// TwinCAT 3 PLC project green_crane
// ProgramVersion: 3.1.4026.19
// libraries:
//   Tc2_Standard, * (Beckhoff Automation GmbH)
//   Tc2_System, * (Beckhoff Automation GmbH)
// project tree:
//   Control/ AB_baseController.TcPOU, FB_AutoControl.TcPOU, FB_manualControl.TcPOU, I_craneControl.TcIO
//   DUTs/ E_CraneModes.TcDUT, E_CraneStatus.TcDUT
//   IOinterface/ FB_ioSim.TcPOU, I_ioInterface.TcIO
//   / PlcTask.TcTTO, simTask.TcTTO
//   POUs/ F_CalcAngle.TcPOU, F_stateMachine.TcPOU, MAIN.TcPOU, ST_inputs_analog.TcDUT, ST_in_digital.TcDUT, ST_ValvePos.TcDUT
//   Simulator/ FB_CylinderSimulator.TcPOU, P_Simulator.TcPOU
// real-time tasks:
//   TASK PlcTask: cycle T#10ms, priority 20, ADS port 350
//   TASK simTask: cycle T#100us, priority 1, ADS port 351

CONFIGURATION green_crane
    RESOURCE PLC ON TwinCAT3
        TASK PlcTask(INTERVAL := T#10ms, PRIORITY := 20);
        TASK simTask(INTERVAL := T#100us, PRIORITY := 1);
        PROGRAM MAIN WITH PlcTask : MAIN;
        PROGRAM P_Simulator WITH simTask : P_Simulator;
    END_RESOURCE
END_CONFIGURATION

// ---- DUTs/E_CraneModes.TcDUT
{attribute 'qualified_only'}
{attribute 'strict'}
{attribute 'to_string'}
TYPE E_CraneModes :
(
	Manual := 0,
	Auto := 1
);
END_TYPE

// ---- DUTs/E_CraneStatus.TcDUT
{attribute 'qualified_only'}
{attribute 'strict'}
{attribute 'to_string'}
TYPE E_CraneStatus :
(
	Off := 0,
	On := 1,
	Ready := 2,
	Running := 3
);
END_TYPE

// ---- POUs/ST_inputs_analog.TcDUT
TYPE ST_inputs_analog :
STRUCT	
	fJoystick : LREAL;
	fPistonPos : LREAL; // [mm] crane piston position
	fP_piston : LREAL; // [bar]
	fP_rod : LREAL; // [bar]
END_STRUCT
END_TYPE

// ---- POUs/ST_in_digital.TcDUT
TYPE ST_in_digital :
STRUCT
	bCranePower : BOOL := FALSE;
	bStartCrane : BOOL := FALSE;
	bEnableCraneMotion : BOOL := FALSE;
	eModeSwitch : E_CraneModes;
END_STRUCT
END_TYPE

// ---- POUs/ST_ValvePos.TcDUT
TYPE ST_ValvePos :
STRUCT
	rCylinderValve : REAL;
END_STRUCT
END_TYPE

// ---- Control/I_craneControl.TcIO
INTERFACE I_craneControl
VAR_INPUT
END_VAR
VAR_OUTPUT
END_VAR

METHOD control_crane
VAR_INPUT
	stInputs : ST_inputs_analog;
END_VAR
VAR_OUTPUT
	fCylValve : REAL;
END_VAR
END_METHOD

METHOD controller
VAR_INPUT
	stButtonInputs : ST_in_digital;
	stAnalogInputs : ST_inputs_analog;
END_VAR
VAR_OUTPUT
	stOutput : ST_ValvePos;
END_VAR
END_METHOD

END_INTERFACE

// ---- IOinterface/I_ioInterface.TcIO
INTERFACE I_ioInterface

METHOD getOutputs
VAR_IN_OUT
	stSimOut : ST_inputs_analog;
END_VAR
END_METHOD

METHOD setInputs
VAR_INPUT
	stValvePos	: ST_ValvePos;
	eCraneState : E_CraneStatus;
END_VAR
END_METHOD

END_INTERFACE

// ---- POUs/MAIN.TcPOU
PROGRAM MAIN
VAR
	stButtonInputs : ST_in_digital;
	stAnalogInputs : ST_inputs_analog;
	stOutputs : ST_ValvePos;
	eCraneMode : E_CraneStatus;
	ipControlMode : I_craneControl;
	fbManual : FB_manualControl;
	fbAuto : FB_AutoControl;
	stValveOut : ST_ValvePos;
	fbIOsim : FB_ioSim;
	fBoomAng : LREAL;
	fBoomAngRef : LREAL;
END_VAR

eCraneMode := F_stateMachine(stButtonInputs);
CASE stButtonInputs.eModeSwitch OF //polymorphism using interface pointer ipControlMode
		E_CraneModes.Manual:
			ipControlMode := fbManual;
		E_CraneModes.Auto:
			ipControlMode := fbAuto;
END_CASE

IF eCraneMode = E_CraneStatus.Running AND ipControlMode <> 0  THEN
	fbIOsim.getOutputs(stSimOut := stAnalogInputs);
	ipControlMode.controller(stButtonInputs := stButtonInputs,
		stAnalogInputs := stAnalogInputs,
		stOutput => stValveOut);
	fbIOsim.setInputs(stValvePos := stValveOut,
		eCraneState := eCraneMode);
END_IF

fBoomAng := F_CalcAngle(stAnalogInputs.fPistonPos);

END_PROGRAM

// ---- Control/FB_manualControl.TcPOU
FUNCTION_BLOCK FB_manualControl EXTENDS AB_baseController
VAR_INPUT
END_VAR
VAR_OUTPUT
END_VAR
VAR
END_VAR

METHOD control_winch
VAR_INPUT
	stInputs	: ST_inputs_analog;
END_VAR
VAR_OUTPUT
	fMotorValve	: REAL;
END_VAR
fMotorValve := -1.0;
END_METHOD

END_FUNCTION_BLOCK

// ---- Control/AB_baseController.TcPOU
FUNCTION_BLOCK ABSTRACT AB_baseController IMPLEMENTS I_craneControl
VAR_INPUT
END_VAR
VAR_OUTPUT
END_VAR
VAR
END_VAR

METHOD ABSTRACT control_crane 
VAR_INPUT
	stInputs	: ST_inputs_analog;
END_VAR
VAR_OUTPUT
	fCylValve	: REAL;
END_VAR
END_METHOD

METHOD controller
VAR_INPUT
	stButtonInputs	: ST_in_digital;
	stAnalogInputs	: ST_inputs_analog;
END_VAR
VAR_OUTPUT
	stOutput	: ST_ValvePos;
END_VAR
stOutput.rCylinderValve := control_crane(stInputs := stAnalogInputs);
END_METHOD

END_FUNCTION_BLOCK

// ---- Control/FB_AutoControl.TcPOU
FUNCTION_BLOCK FB_AutoControl EXTENDS AB_baseController
VAR_INPUT
END_VAR
VAR_OUTPUT
END_VAR
VAR
END_VAR

METHOD control_crane
VAR_INPUT
	stInputs	: ST_inputs_analog;
END_VAR
VAR_OUTPUT
	fCylValve	: REAL;
END_VAR
fCylValve := 0;
END_METHOD

END_FUNCTION_BLOCK

// ---- IOinterface/FB_ioSim.TcPOU
FUNCTION_BLOCK PUBLIC FB_ioSim IMPLEMENTS I_ioInterface
VAR_INPUT
END_VAR
VAR_OUTPUT
END_VAR
VAR
END_VAR

METHOD getOutputs
VAR_IN_OUT
	stSimOut : ST_inputs_analog;
END_VAR
stSimOut.fP_piston := P_Simulator.stSimSystemOutputs.fP_piston;
stSimOut.fP_rod := P_Simulator.stSimSystemOutputs.fP_rod;
stSimOut.fPistonPos := P_Simulator.stSimSystemOutputs.fPistonPos;
END_METHOD

METHOD setInputs
VAR_INPUT
	stValvePos	: ST_ValvePos;
	eCraneState	: E_CraneStatus;
END_VAR
P_Simulator.stSimInputs := stValvePos;
P_Simulator.eCraneState := eCraneState;
END_METHOD

END_FUNCTION_BLOCK

// ---- Simulator/P_Simulator.TcPOU
PROGRAM P_Simulator
VAR
	fbCylinderSim : FB_CylinderSimulator;
END_VAR
VAR_INPUT
	stSimSystemOutputs : ST_inputs_analog;
	eCraneState : E_CraneStatus;
	stSimInputs : ST_ValvePos;
END_VAR

IF eCraneState <> E_CraneStatus.Off THEN // <> = !=
	fbCylinderSim(ssMethodType := 1,
		fNormalizedValveInput := stSimInputs.rCylinderValve,
		fPistonPosition_m => stSimSystemOutputs.fPistonPos,
		fPistonSidePressure_bar => stSimSystemOutputs.fP_piston,
		fRodSidePressure_bar => stSimSystemOutputs.fP_rod);
ELSE
	fbCylinderSim(ssMethodType := 0);
END_IF

END_PROGRAM

// ---- Simulator/FB_CylinderSimulator.TcPOU
FUNCTION_BLOCK FB_CylinderSimulator
VAR_INPUT
	ssMethodType: SINT;
	fNormalizedValveInput: LREAL;
END_VAR
VAR_OUTPUT
	fPistonPosition_m: LREAL;
	fPistonSidePressure_bar: LREAL;
	fRodSidePressure_bar: LREAL;
END_VAR
VAR
	pLS: LREAL;
	QDCV_out: LREAL;
	rtb_xDot: LREAL;
	rtb_xDotDot: LREAL;
	y: DINT;
	temp1: LREAL;
	temp2: LREAL;
	temp3: LREAL;
	temp4: LREAL;
	c_DiscreteTimeIntegrator2_D: LREAL;
	c_DiscreteTimeIntegrator3_D: LREAL;
	c_DiscreteTimeIntegrator_DS: LREAL;
	c_DiscreteTimeIntegrator4_D: LREAL;
END_VAR



CASE ssMethodType OF
    0: 
        (* SystemInitialize for Atomic SubSystem: '<Root>/FB_CylinderSimulator' *)
        (* InitializeConditions for DiscreteIntegrator: '<S1>/Discrete-Time Integrator' *)
        c_DiscreteTimeIntegrator_DS := 6.874E+6;
        (* InitializeConditions for DiscreteIntegrator: '<S1>/Discrete-Time Integrator2' *)
        c_DiscreteTimeIntegrator2_D := 0.0;
        (* InitializeConditions for DiscreteIntegrator: '<S1>/Discrete-Time Integrator3' *)
        c_DiscreteTimeIntegrator3_D := 0.0;
        (* InitializeConditions for DiscreteIntegrator: '<S1>/Discrete-Time Integrator4' *)
        c_DiscreteTimeIntegrator4_D := 514400.0;
        (* End of SystemInitialize for SubSystem: '<Root>/FB_CylinderSimulator' *)
    1: 
        (* Outputs for Atomic SubSystem: '<Root>/FB_CylinderSimulator' *)
        (* DiscreteIntegrator: '<S1>/Discrete-Time Integrator2' *)
        rtb_xDot := c_DiscreteTimeIntegrator2_D;
        (* Outport: '<Root>/fPistonPosition_m' incorporates:
         *  DiscreteIntegrator: '<S1>/Discrete-Time Integrator3' *)
        fPistonPosition_m := c_DiscreteTimeIntegrator3_D;
        (* Outport: '<Root>/fPistonSidePressure_bar' incorporates:
         *  DiscreteIntegrator: '<S1>/Discrete-Time Integrator'
         *  Gain: '<S1>/Gain' *)
        fPistonSidePressure_bar := 1.0E-5 * c_DiscreteTimeIntegrator_DS;
        (* Outport: '<Root>/fRodSidePressure_bar' incorporates:
         *  DiscreteIntegrator: '<S1>/Discrete-Time Integrator4'
         *  Gain: '<S1>/Gain1' *)
        fRodSidePressure_bar := 1.0E-5 * c_DiscreteTimeIntegrator4_D;
        (* MATLAB Function: '<S1>/MATLAB Function' incorporates:
         *  DiscreteIntegrator: '<S1>/Discrete-Time Integrator'
         *  DiscreteIntegrator: '<S1>/Discrete-Time Integrator2'
         *  DiscreteIntegrator: '<S1>/Discrete-Time Integrator3'
         *  DiscreteIntegrator: '<S1>/Discrete-Time Integrator4' *)
        (* Parameters *)
        (* MATLAB Function 'FB_CylinderSimulator/MATLAB Function': '<S2>:1' *)
        (* '<S2>:1:3' mEffective = 1.5e+04; *)
        (* [kg] *)
        (* '<S2>:1:4' Fexternal = 2.15e+04; *)
        (* [N] *)
        (* '<S2>:1:5' kFric = 10000; *)
        (* [N/(ms)] *)
        (* '<S2>:1:6' Apiston = 0.0033; *)
        (* [m^2] *)
        (* '<S2>:1:7' Aannulus = 0.0023; *)
        (* [m^2] *)
        (* '<S2>:1:8' beta = 1.0e9; *)
        (* [Pa] *)
        (* '<S2>:1:9' pSupply = 180e5; *)
        (* [Pa] *)
        (* '<S2>:1:10' pReturn = 1.1e5; *)
        (* [Pa] *)
        (* '<S2>:1:11' MaxStroke = 0.5; *)
        (* [m] *)
        (* '<S2>:1:12' VCyl_A = 1.0e-03; *)
        (* '<S2>:1:13' VCyl_B = 1.25e-03; *)
        (* '<S2>:1:14' p_nom_DCV = 7e5; *)
        (* '<S2>:1:15' Q1_ref_DCV = 20/6e4; *)
        (* '<S2>:1:16' Q2_ref_DCV = 8/6e4; *)
        (* '<S2>:1:17' kv1_DCV = Q1_ref_DCV/sqrt(p_nom_DCV); *)
        (* '<S2>:1:18' kv2_DCV = Q2_ref_DCV/sqrt(p_nom_DCV); *)
        (* '<S2>:1:19' p0 = 7e5; *)
        (* compensator crack pressure *)
        (* Directional Control Valve - Lifting Cylinder  *)
        (* LS Pressure *)
        (* '<S2>:1:22' if uDCV > 0 *)

        IF fNormalizedValveInput > 0.0 THEN 
            (* '<S2>:1:23' pLS = pPiston; *)
            pLS := c_DiscreteTimeIntegrator_DS;
        ELSIF fNormalizedValveInput < 0.0 THEN 
            (* '<S2>:1:24' elseif uDCV < 0 *)
            (* '<S2>:1:25' pLS = pRod; *)
            pLS := c_DiscreteTimeIntegrator4_D;
        ELSE 
            (* '<S2>:1:26' else *)
            (* '<S2>:1:27' pLS = 0; *)
            pLS := 0.0;
        END_IF;

        (* '<S2>:1:30' if pLS<0 *)

        IF pLS < 0.0 THEN 
            (* '<S2>:1:31' pLS = 0; *)
            pLS := 0.0;
        END_IF;

        (* Pressure Compensator *)
        (* '<S2>:1:35' pPC = 0; *)
        (* '<S2>:1:37' if p0 <= (pSupply - pLS) *)

        IF (1.8E+7 - pLS) >= 700000.0 THEN 
            (* '<S2>:1:38' pPC = pLS+p0; *)
            pLS := pLS + 700000.0;
        ELSE 
            (* '<S2>:1:39' elseif 0 < (pSupply - pLS) < p0 *)
            (* '<S2>:1:40' pPC = pSupply-pLS; *)
            pLS := 1.8E+7 - pLS;
        END_IF;

        (* '<S2>:1:45' if pPC<0 *)

        IF pLS < 0.0 THEN 
            (* '<S2>:1:46' pPC = 0; *)
            pLS := 0.0;
        END_IF;

        (* Orifice Equations *)
        (* '<S2>:1:49' if uDCV > 0 *)

        IF fNormalizedValveInput > 0.0 THEN 
            (* '<S2>:1:50' QDCV_in =  kv1_DCV*uDCV*sign(pPC-pPiston)*sqrt(abs(pPC-pPiston)); *)
            pLS := pLS - c_DiscreteTimeIntegrator_DS;

            IF pLS < 0.0 THEN 
                y := -1;
            ELSIF pLS > 0.0 THEN 
                y := 1;
            ELSE 
                y := 0;
            END_IF;

            temp3 := ABS(pLS);
            pLS := ((3.9840953644479785E-7 * fNormalizedValveInput) * DINT_TO_LREAL(y)) * SQRT(temp3);
            (* QpistonSide *)
            (* '<S2>:1:51' QDCV_out = kv2_DCV*uDCV*sign(pRod-pReturn)*sqrt(abs(pRod-pReturn)); *)

            IF (c_DiscreteTimeIntegrator4_D - 110000.0) < 0.0 THEN 
                y := -1;
            ELSIF (c_DiscreteTimeIntegrator4_D - 110000.0) > 0.0 THEN 
                y := 1;
            ELSE 
                y := 0;
            END_IF;

            temp4 := ABS(c_DiscreteTimeIntegrator4_D - 110000.0);
            QDCV_out := ((1.5936381457791916E-7 * fNormalizedValveInput) * DINT_TO_LREAL(y)) * SQRT(temp4);
            (* QrodSide *)
        ELSIF fNormalizedValveInput < 0.0 THEN 
            (* '<S2>:1:52' elseif uDCV < 0 *)
            (* '<S2>:1:53' QDCV_out =  kv1_DCV*uDCV*sign(pPC-pRod)*sqrt(abs(pPC-pRod)); *)
            pLS := pLS - c_DiscreteTimeIntegrator4_D;

            IF pLS < 0.0 THEN 
                y := -1;
            ELSIF pLS > 0.0 THEN 
                y := 1;
            ELSE 
                y := 0;
            END_IF;

            temp1 := ABS(pLS);
            QDCV_out := ((3.9840953644479785E-7 * fNormalizedValveInput) * DINT_TO_LREAL(y)) * SQRT(temp1);
            (* QrodSide *)
            (* '<S2>:1:54' QDCV_in =  kv2_DCV*uDCV*sign(pPiston-pReturn)*sqrt(abs(pPiston-pReturn)); *)

            IF (c_DiscreteTimeIntegrator_DS - 110000.0) < 0.0 THEN 
                y := -1;
            ELSIF (c_DiscreteTimeIntegrator_DS - 110000.0) > 0.0 THEN 
                y := 1;
            ELSE 
                y := 0;
            END_IF;

            temp2 := ABS(c_DiscreteTimeIntegrator_DS - 110000.0);
            pLS := ((1.5936381457791916E-7 * fNormalizedValveInput) * DINT_TO_LREAL(y)) * SQRT(temp2);
            (* QpistonSide *)
        ELSE 
            (* '<S2>:1:55' else *)
            (* '<S2>:1:56' QDCV_in = 0; *)
            pLS := 0.0;
            (* '<S2>:1:57' QDCV_out = 0; *)
            QDCV_out := 0.0;
        END_IF;

        (* Pressure Gradients *)
        (* '<S2>:1:60' VA = VCyl_A + x*Apiston; *)
        (* '<S2>:1:61' VB =  VCyl_B + (MaxStroke - x)*Aannulus; *)
        (* '<S2>:1:62' VA_dot = Apiston*xDot; *)
        (* '<S2>:1:63' VB_dot = Aannulus*xDot; *)
        (* '<S2>:1:64' pPistonDot = beta/VA*(QDCV_in - VA_dot); *)
        (* '<S2>:1:65' pRodDot = beta/VB*(VB_dot-QDCV_out); *)
        QDCV_out := (1.0E+9 / (((0.5 - c_DiscreteTimeIntegrator3_D) * 0.0023) + 0.00125)) * ((0.0023 * c_DiscreteTimeIntegrator2_D) - QDCV_out);
        (* Viscouse Friction *)
        (* '<S2>:1:68' Ffric = kFric*xDot; *)
        (* Hydraulic Force *)
        (* '<S2>:1:70' Fhyd = pPiston*Apiston - pRod*Aannulus; *)
        (* Newton Second Law of Motion *)
        (* '<S2>:1:73' xDotDot = (Fhyd - Ffric - Fexternal)/mEffective; *)
        rtb_xDotDot := ((((c_DiscreteTimeIntegrator_DS * 0.0033) - (c_DiscreteTimeIntegrator4_D * 0.0023)) - (10000.0 * c_DiscreteTimeIntegrator2_D)) - 21500.0) / 15000.0;
        (* Update for DiscreteIntegrator: '<S1>/Discrete-Time Integrator' incorporates:
         *  DiscreteIntegrator: '<S1>/Discrete-Time Integrator2'
         *  DiscreteIntegrator: '<S1>/Discrete-Time Integrator3'
         *  MATLAB Function: '<S1>/MATLAB Function' *)
        c_DiscreteTimeIntegrator_DS := (((1.0E+9 / ((c_DiscreteTimeIntegrator3_D * 0.0033) + 0.001)) * (pLS - (0.0033 * c_DiscreteTimeIntegrator2_D))) * 0.0001) + c_DiscreteTimeIntegrator_DS;

        IF c_DiscreteTimeIntegrator_DS > 1.8E+7 THEN 
            c_DiscreteTimeIntegrator_DS := 1.8E+7;
        ELSIF c_DiscreteTimeIntegrator_DS < 110000.0 THEN 
            c_DiscreteTimeIntegrator_DS := 110000.0;
        END_IF;

        (* End of Update for DiscreteIntegrator: '<S1>/Discrete-Time Integrator' *)
        

        (* Update for DiscreteIntegrator: '<S1>/Discrete-Time Integrator2' *)
        c_DiscreteTimeIntegrator2_D := (0.0001 * rtb_xDotDot) + c_DiscreteTimeIntegrator2_D;
        (* Update for DiscreteIntegrator: '<S1>/Discrete-Time Integrator3' *)
        c_DiscreteTimeIntegrator3_D := (0.0001 * rtb_xDot) + c_DiscreteTimeIntegrator3_D;

        IF c_DiscreteTimeIntegrator3_D > 0.5 THEN 
            c_DiscreteTimeIntegrator3_D := 0.5;
        ELSIF c_DiscreteTimeIntegrator3_D < 0.0 THEN 
            c_DiscreteTimeIntegrator3_D := 0.0;
        END_IF;

        (* End of Update for DiscreteIntegrator: '<S1>/Discrete-Time Integrator3' *)
        

        (* Update for DiscreteIntegrator: '<S1>/Discrete-Time Integrator4' *)
        c_DiscreteTimeIntegrator4_D := (0.0001 * QDCV_out) + c_DiscreteTimeIntegrator4_D;

        IF c_DiscreteTimeIntegrator4_D > 1.8E+7 THEN 
            c_DiscreteTimeIntegrator4_D := 1.8E+7;
        ELSIF c_DiscreteTimeIntegrator4_D < 110000.0 THEN 
            c_DiscreteTimeIntegrator4_D := 110000.0;
        END_IF;

        (* End of Update for DiscreteIntegrator: '<S1>/Discrete-Time Integrator4' *)
        (* End of Outputs for SubSystem: '<Root>/FB_CylinderSimulator' *)
END_CASE;

END_FUNCTION_BLOCK

// ---- POUs/F_stateMachine.TcPOU
FUNCTION F_stateMachine : E_CraneStatus
VAR_INPUT
	stButtonInputs : ST_in_digital;
END_VAR
VAR
	eState : E_CraneStatus;
END_VAR

IF stButtonInputs.bCranePower THEN
	eState := E_CraneStatus.On;
	IF stButtonInputs.bEnableCraneMotion THEN
		eState := E_CraneStatus.Ready;
		IF stButtonInputs.bStartCrane THEN
			eState := E_CraneStatus.Running;
		END_IF
	END_IF
ELSE
	eState := E_CraneStatus.Off;
END_IF
F_stateMachine := eState;

END_FUNCTION

// ---- POUs/F_CalcAngle.TcPOU
FUNCTION F_CalcAngle : LREAL // [rad] output
VAR_INPUT
	xCyl : LREAL; // [m] cylinder position
END_VAR
VAR
	ABx : LREAL := 0.427;
	ABy : LREAL := 1.057;
	ACx : LREAL := 0.49484;
	ACy : LREAL := 0.133;
	
	AB : LREAL;
	AC : LREAL;
	BC : LREAL;
	alpha1 : LREAL;
	alpha2 : LREAL;
END_VAR

AB := SQRT(EXPT(ABS(ABx),2) + EXPT(ABS(ABy),2));
AC := SQRT(EXPT(ABS(ACx),2) + EXPT(ABS(ACy),2));

BC := 0.77222 + xCyl;

alpha1 := ATAN(ABS(ACy)/ABS(ACx));
alpha2 := ATAN(ABS(ABy)/ABS(ABx));

F_CalcAngle := ACOS( (EXPT(ABS(AB),2) + EXPT(ABS(AC),2) - (EXPT(ABS(BC),2))) / (2 * ABS(AB)*ABS(AC)) ) - alpha1 + alpha2;

END_FUNCTION
